(* IEC 61131-3 sources: PLC_02/ArCan1/ArCanReceive, 2 files *)

(* ---- ArCanReceive.typ ---- *)
TYPE
	ArCanReceive_steps :
		(
		STEP_ERROR := 255,
		STEP_DEINIT := 254,
		STEP_WAIT_FOR_DATA := 10,
		STEP_INIT_RECEIVER := 2,
		STEP_INIT_BAUDRATE := 1,
		STEP_WAIT := 0
		);
	ArCanReceive_typ : 	STRUCT
		step : ArCanReceive_steps := STEP_WAIT;
		ArCanSetBitTimingRegisters_0 : ArCanSetBitTimingRegisters;
		ArCanReceiver_0 : ArCanReceive;
		receiverDeviceName : STRING[80];
		receivedIterationCounter : UDINT;
		lastReceiveTimestamp : UDINT;
		lostFrames : UDINT;
		successCount : UDINT;
		errorCount : UINT;
		lastError : DINT;
		enable : BOOL;
		id : UDINT;
		idMask : UDINT;
		format : UDINT;
		queueSize : UDINT;
	END_STRUCT;
END_TYPE

(* ---- ArCanReceive.st ---- *)
// CAN_CH_B

PROGRAM _INIT
	RackSyS;
	ActArCanReceiver;
	ArCanReceiver.enable				:= TRUE;
	ArCanReceiver.receiverDeviceName 	:= 'IF6.ST1.IF1';       (* for X20CP0482 CPU *)
	ArCanReceiver.id					:= 0;
	ArCanReceiver.idMask				:= arCAN_RECEIVE_ALL;  // or configure IDMask
	ArCanReceiver.format				:= arCAN_11BIT;  // or arCAN_29BIT
	ArCanReceiver.queueSize				:= 128;
	ArCanReceiver.ArCanSetBitTimingRegisters_0.Register0 := 16#00;
	ArCanReceiver.ArCanSetBitTimingRegisters_0.Register1 := 16#1C;

	(**********************	 CAN Baud rate Register Value	*************************)
	(********************************************************************************)
	(* 	  1 000 000 bit/s    >>		Register0 = 16#00	||		Register1 = 16#14	*)
	(* 		800 000 bit/s    >>		Register0 = 16#00	||		Register1 = 16#16	*)
	(* 		500 000 bit/s    >>		Register0 = 16#00	||		Register1 = 16#1C	*)
	(* 		250 000 bit/s    >>		Register0 = 16#01	||		Register1 = 16#1C	*)
	(* 		125 000 bit/s    >>		Register0 = 16#03	||		Register1 = 16#1C	*)
	(* 		100 000 bit/s    >>		Register0 = 16#04	||		Register1 = 16#1C	*)
	(* 		050 000 bit/s    >>		Register0 = 16#09	||		Register1 = 16#1C	*)
	(* 		020 000 bit/s    >>		Register0 = 16#18	||		Register1 = 16#1C	*)
	(* 		010 000 bit/s    >>		Register0 = 16#31	||		Register1 = 16#1C	*)
	(********************************************************************************)
	(********************************************************************************)

END_PROGRAM

PROGRAM _CYCLIC
//	RackSyS[0].RackIro
	(* Action for ArCanReceiver *)
	ActArCanReceiver;
	(***********************************************************)
	(* Customize the received data *)
	// ArCanReceiver.ArCanReceiver_0.ReceivedFrame; //Data received
	IF (ArCanReceiver.ArCanReceiver_0.NewDataValid) THEN

		CASE ArCanReceiver.ArCanReceiver_0.ReceivedFrame.ID OF
			16#500..16#510:
			Can1[0].Count := Can1[0].Count +1;
			IF  Can1[0].Count	>=3600 THEN
				Can1[0].Count :=0;
			END_IF;

			IF ArCanReceiver.ArCanReceiver_0.ReceivedFrame.ID = 16#500 THEN
				Can[2].CanInfoArry[0]   := SHL(BYTE_TO_UINT(ArCanReceiver.ArCanReceiver_0.ReceivedFrame.Data[1]),8)OR BYTE_TO_UINT(ArCanReceiver.ArCanReceiver_0.ReceivedFrame.Data[0]);
				Can[2].CanInfoArry[1] 	:= SHL(BYTE_TO_UINT(ArCanReceiver.ArCanReceiver_0.ReceivedFrame.Data[3]),8)OR BYTE_TO_UINT(ArCanReceiver.ArCanReceiver_0.ReceivedFrame.Data[2]);
				Can[2].CanInfoArry[2] 	:= SHL(BYTE_TO_UINT(ArCanReceiver.ArCanReceiver_0.ReceivedFrame.Data[5]),8)OR BYTE_TO_UINT(ArCanReceiver.ArCanReceiver_0.ReceivedFrame.Data[4]);
				Can[2].CanInfoArry[3]	:= SHL(BYTE_TO_UINT(ArCanReceiver.ArCanReceiver_0.ReceivedFrame.Data[7]),8)OR BYTE_TO_UINT(ArCanReceiver.ArCanReceiver_0.ReceivedFrame.Data[6]);
			END_IF;
			IF ArCanReceiver.ArCanReceiver_0.ReceivedFrame.ID = 16#501 THEN
				Can[3].CanInfoArry[0]   := SHL(BYTE_TO_UINT(ArCanReceiver.ArCanReceiver_0.ReceivedFrame.Data[1]),8)OR BYTE_TO_UINT(ArCanReceiver.ArCanReceiver_0.ReceivedFrame.Data[0]);
				Can[3].CanInfoArry[1] 	:= SHL(BYTE_TO_UINT(ArCanReceiver.ArCanReceiver_0.ReceivedFrame.Data[3]),8)OR BYTE_TO_UINT(ArCanReceiver.ArCanReceiver_0.ReceivedFrame.Data[2]);
				Can[3].CanInfoArry[2] 	:= SHL(BYTE_TO_UINT(ArCanReceiver.ArCanReceiver_0.ReceivedFrame.Data[5]),8)OR BYTE_TO_UINT(ArCanReceiver.ArCanReceiver_0.ReceivedFrame.Data[4]);
				Can[3].CanInfoArry[3]	:= SHL(BYTE_TO_UINT(ArCanReceiver.ArCanReceiver_0.ReceivedFrame.Data[7]),8)OR BYTE_TO_UINT(ArCanReceiver.ArCanReceiver_0.ReceivedFrame.Data[6]);
			END_IF;
//			16#06080000..16#06080008:
//			RackSyS[1].RackCanCount := RackSyS[1].RackCanCount +1;
//			16#620..16#62E:
//			RackSyS[2].RackCanCount := RackSyS[2].RackCanCount +1;
//			16#630..16#63E:
//			RackSyS[3].RackCanCount := RackSyS[3].RackCanCount +1;
			//Can_DB_Key.Header	:=  UDINT_TO_USINT(ArCanReceiver.ArCanReceiver_0.ReceivedFrame.ID - 16#600)/16;
			//Can_DB_Key.Body		:= 	UDINT_TO_USINT(ArCanReceiver.ArCanReceiver_0.ReceivedFrame.ID - 16#600)-Can_DB_Key.Header*16;
			// memcpy(ADR(Can_Data[Can_DB_Key.Header].r6N[Can_DB_Key.Body]),ADR(ArCanReceiver.ArCanReceiver_0.ReceivedFrame.Data),8);
		END_CASE;

	END_IF

	//	IF ArCanReceiver.ArCanReceiver_0.ReceivedFrame.ID = 16#CanID THEN
	//		memcpy(ADR(TargetVariable), ADR(ArCanReceiver.ArCanReceiver_0.ReceivedFrame.Data), SIZEOF(ArCanReceiver.ArCanReceiver_0.ReceivedFrame.DataLength));
	//	ELSIF ArCanReceiver.ArCanReceiver_0.ReceivedFrame.ID = 16#CanID THEN
	//		memcpy(ADR(TargetVariable), ADR(ArCanReceiver.ArCanReceiver_0.ReceivedFrame.Data), SIZEOF(ArCanReceiver.ArCanReceiver_0.ReceivedFrame.DataLength));
	//	END_IF

	(***********************************************************)
	(* CAN Communication Status *)
	(***********************************************************)

	IF ArCanReceiver.ArCanReceiver_0.Error THEN
		gComm.CAN1.bError	:= TRUE;
		gComm.CAN1.bActive	:= FALSE;
		gComm.CAN1.bTransmitting	:= FALSE;
	ELSIF ArCanReceiver.ArCanReceiver_0.Active AND ArCanReceiver.ArCanReceiver_0.Busy THEN
		gComm.CAN1.bError	:= FALSE;
		gComm.CAN1.bActive	:= TRUE;

		IF (countCANSuccessOld <> ArCanReceiver.successCount) THEN
			countCANSuccessOld	:= ArCanReceiver.successCount;
			gComm.CAN1.bTransmitting	:= TRUE;
			countTime	:= 0;
		ELSE
			countTime	:= countTime + 1;
			IF (countTime > 50) THEN
				gComm.CAN1.bTransmitting	:= FALSE;
				countTime	:= 0;
			END_IF
		END_IF
	ELSE
		gComm.CAN1.bError	:= FALSE;
		gComm.CAN1.bActive	:= FALSE;
		gComm.CAN1.bTransmitting	:= FALSE;
	END_IF
	(***********************************************************)

END_PROGRAM

PROGRAM _EXIT

	(* Deinitialization of the receiver *)
	ArCanReceiver.ArCanReceiver_0.Enable	:= FALSE;
	ArCanReceiver.ArCanReceiver_0();

END_PROGRAM
